// TIA Portal V17 export
// export: Created 2025-03-07T09:19:21.5668318Z, ExportSetting WithDefaults, DisplayName Totally Integrated Automation Portal, DisplayVersion V17 Update 8, DisplayName TIA Portal Openness, DisplayVersion V17 Update 8, DisplayName TIA Portal Version Control Interface, DisplayVersion V17, DisplayName SINAMICS Startdrive Advanced, DisplayVersion V17 SP2, DisplayName SINAMICS Startdrive G110M, G120, G120C, G120D, G120P, G115D, DisplayVersion V17 SP2, DisplayName SINAMICS Startdrive G130, G150, S120, S150, SINAMICS MV, S210, DisplayVersion V17 SP2, DisplayName STEP 7 Professional, DisplayVersion V17 Update 8, DisplayName SINUMERIK ONE STEP 7 Toolbox, DisplayVersion V17 Update 12, DisplayName SINUMERIK 840D sl STEP 7 Toolbox, DisplayVersion V17 Update 12, DisplayName STEP 7 Safety, DisplayVersion V17 Update 6, DisplayName WinCC Advanced, DisplayVersion V17 Update 8
VAR_GLOBAL   // PLC tag table "Default tag table"
   UNIT_01_STA_1_CYCLE_AUTO_REQ AT %T120 : Timer;
   UNIT_02_STA_0_CYCLE_AUTO_REQ AT %T528 : Timer;
   UNIT_02_STA_1_CYCLE_AUTO_REQ AT %T121 : Timer;
   UNIT_01_STA_0_CYCLE_AUTO_REQ AT %T529 : Timer;
   DUMMY_M70 AT %M70.0 : Bool;
   UNIT_02_ASPIRATION_LOW_WARNING_TIMER AT %T536 : Timer;
   UNIT_01_ASPIRATION_HIGH_ALARM_TIMER AT %T531 : Timer;
   UNIT_02_ASPIRATION_HIGH_WARNING_TIMER AT %T537 : Timer;
   UNIT_02_ASPIRATION_HIGH_ALARM_TIMER AT %T535 : Timer;
   UNIT_01_ASPIRATION_LOW_ALARM_TIMER AT %T530 : Timer;
   UNIT_01_ASPIRATION_LOW_WARNING_TIMER AT %T532 : Timer;
   UNIT_01_ASPIRATION_HIGH_WARNING_TIMER AT %T533 : Timer;
   UNIT_02_ASPIRATION_LOW_ALARM_TIMER AT %T534 : Timer;
   Tag_3 AT %M700.2 : Bool;
   Tag_2 AT %M700.1 : Bool;
   Tag_1 AT %M70.5 : Bool;
   CELL_DOOR_CLOSED AT %M5.7 : Bool;   // CELL DOOR CLOSED
   Tag_4 AT %M700.3 : Bool;
   GENERAL_GAS_PNEUM_SYS_Q AT %Q50.2 : Bool;   // GENERAL GAS PNEUMATIC SYSTEM ON OUTPUT
   UNIT_01_PROTEC_GAS_SW_OFF_Q AT %Q71.4 : Bool;
   M60_POWDER_STABILIZATION_ACK_DELAY_TIMER AT %T256 : Timer;
   M60_POWDER_STABILIZATION_U02_ACK_DELAY_TIMER AT %T257 : Timer;
   STATION_3_LIGHT_U01_Q AT %Q33.2 : Bool;   // STATION 3 LIGHT UNIT 01 OUTPUT
   STATION_3_LIGHT_U02_Q AT %Q33.3 : Bool;   // STATION 3 LIGHT UNIT 02 OUTPUT
   U02_TURCK_HOME_Q AT %Q1606.7 : Bool;   // UNIT 02 BIMANUAL HOME OUTPUT
   U02_TURCK_RESET_FAULTS_I AT %I1606.4 : Bool;   // UNIT 02 BIMANUAL RESET FAULTS INPUT
   U02_TURCK_RESET_FAULTS_Q AT %Q1606.5 : Bool;   // UNIT 02 BIMANUAL RESET FAULTS OUTPUT
   U02_TURCK_UNLD_PART_Q AT %Q1606.1 : Bool;   // UNIT 02 BIMANUAL UNLOADED PART OUTPUT
   U02_TURCK_UNLD_PART_I AT %I1606.0 : Bool;   // UNIT 02 BIMANUAL UNLOAD PART INPUT
   U02_TURCK_HOME_I AT %I1606.6 : Bool;   // UNIT 02 BIMANUAL HOME INPUT
   U02_TURCK_LD_PART_I AT %I1606.2 : Bool;   // UNIT 02 BIMANUAL LOAD PART INPUT
   U02_TURCK_LD_PART_Q AT %Q1606.3 : Bool;   // UNIT 02 BIMANUAL LOADED PART OUTPUT
   Tag_5 AT %I690.4 : Bool;
   Tag_6 AT %M568.6 : Bool;
   Tag_7 AT %M70.1 : Bool;
   Tag_8 AT %M80.4 : Bool;
   Tag_10 AT %M77.6 : Bool;
   Tag_9 AT %M77.7 : Bool;
   Tag_11 AT %Q1066.6 : Bool;
   Tag_13 AT %Q1067.0 : Bool;
   Tag_12 AT %Q1066.7 : Bool;
   Tag_14 AT %T259 : Timer;
   Tag_57 AT %T258 : Timer;
   TIMER_PRUEBA AT %T96 : Timer;
   Tag_15 AT %T1501 : Timer;
   U01_ASPIRATION_PRESSURE_VALUE AT %IW550 : Word;
   U02_ASPIRATION_PRESSURE_VALUE AT %IW552 : Word;
   Tag_16 AT %M69.0 : Bool;
   Tag_17 AT %MW400 : Int;
   Tag_18 AT %M69.1 : Bool;
   Tag_19 AT %I1690.0 : Bool;
   Tag_20 AT %MW452 : Int;
END_VAR
